// TIA Portal V20 export
TYPE "LER_typeQrData"
// stored: Access Published
   STRUCT
      QrReadOk : Bool;
      QrReadNG : Bool;
      QrReadComplete : Bool;
      QrReadID : String[64];
   END_STRUCT;
END_TYPE
